// TIA Portal V16 export
// export: Created 2026-04-09T13:37:01.5819548Z, ExportSetting WithDefaults, DisplayName Totally Integrated Automation Portal, DisplayVersion V16, DisplayName TIA Portal Version Control Interface, DisplayVersion V16, DisplayName TIA Portal Openness, DisplayVersion V16, DisplayName STEP 7 Professional, DisplayVersion V16, DisplayName STEP 7 Safety, DisplayVersion V16, DisplayName WinCC Advanced, DisplayVersion V16
VAR_GLOBAL   // PLC tag table "Standard-Variablentabelle"
   start AT %I0.4 : Bool;
   sensor1 AT %I0.0 : Bool;
   sensor2 AT %I0.1 : Bool;
   sensor3 AT %I0.2 : Bool;
   stop AT %I0.5 : Bool;
   "emergency stop" AT %I0.3 : Bool;
   "Detect Z" AT %I0.6 : Bool;
   movingx AT %I0.7 : Bool;
   movingz AT %I1.0 : Bool;
   rotating AT %I1.1 : Bool;
   "gripper rotating" AT %I1.2 : Bool;
   belt4m AT %Q0.0 : Bool;
   blet6m1 AT %Q0.1 : Bool;
   belt6m2 AT %Q0.2 : Bool;
   roller4m1 AT %Q0.3 : Bool;
   roller6m1 AT %Q0.4 : Bool;
   roller6m2 AT %Q0.5 : Bool;
   roller4m AT %Q0.6 : Bool;
   "Rob move x" AT %Q0.7 : Bool;
   "Rob move z" AT %Q1.0 : Bool;
   grab AT %Q1.1 : Bool;
   X AT %M0.0 : Bool;
   SBox AT %M0.1 : Bool;
   LBox AT %M0.2 : Bool;
   Pallet AT %M0.3 : Bool;
   Tag_3 AT %M7.0 : Bool;
   incrementer AT %MW1 : Int;
   Tag_1 AT %M7.1 : Bool;
   T1DN AT %M3.0 : Bool;
   T2DN AT %M3.1 : Bool;
   T3DN AT %M3.2 : Bool;
   T4DN AT %M3.3 : Bool;
   T5DN AT %M3.4 : Bool;
   T6DN AT %M3.5 : Bool;
   T7DN AT %M3.6 : Bool;
   T8DN AT %M3.7 : Bool;
   "Move Rollers" AT %M4.0 : Bool;
   Tag_2 AT %M7.2 : Bool;
   "Rob Start" AT %M7.3 : Bool;
   Tag_4 AT %M5.0 : Bool;
   Tag_5 AT %M5.1 : Bool;
   "Repeat cycle" AT %M4.1 : Bool;
   Tag_6 AT %M5.2 : Bool;
   "CYC DN" AT %M5.3 : Bool;
   "CTU1 DN" AT %M5.4 : Bool;
   Tag_7 AT %M5.5 : Bool;
   "Move rollers again" AT %M5.6 : Bool;
   Tag_8 AT %M5.7 : Bool;
   T_CTU1DN AT %M6.0 : Bool;
   "End Pallet" AT %M6.1 : Bool;
   Tag_9 AT %M6.2 : Bool;
   Tag_10 AT %M6.3 : Bool;
   "T0.1DN" AT %M6.4 : Bool;
   TCTDN AT %M6.5 : Bool;
END_VAR
